FUNCTION_BLOCK Test_TStreamAdd_Read_PVOID EXTENDS T_UnitTestBase
VAR
    Stream : T_Stream(StreamLength := 2);
    ArgType : E_ArgTypeId := E_ArgTypeId.Type_PVOID;
    Bob : INT;
END_VAR

Stream.Init(2);

// add a pointer...
Stream.SetNextArgTypeId(ArgType);
Stream.Add_PVOID(ADR(Bob));

Stream.Seek(0);

// check next arg type is correct...
Assertion.AssertEquals_INT(Expected     := ArgType,
                           Actual       := Stream.GetNextArgTypeId(),
                           VariableName := 'Stream.GetNextArgTypeId()');

// check next value...	
Assertion.AssertEquals_PVOID(Expected     := ADR(Bob),
                             Actual       := Stream.Read_PVOID(),
                             VariableName := 'Stream.Read_PVOID()');

// check we are at the end of the stream..							
Assertion.AssertEquals_UDINT(Expected     := Stream.StreamLength,
                             Actual       := Stream.Position,
                             VariableName := 'Stream.Position');

TestFinished();

END_FUNCTION_BLOCK

(* stored: Version 1.1.0.1, ProductVersion 3.1.4024.6
   POU Test_TStreamAdd_Read_PVOID: Id {84951354-6441-44c9-b63c-255267689420}, SpecialFunc None *)
